KUKA KRL program: Robotica_Trabalho_v4.src, Robotica_Trabalho_v4.dat

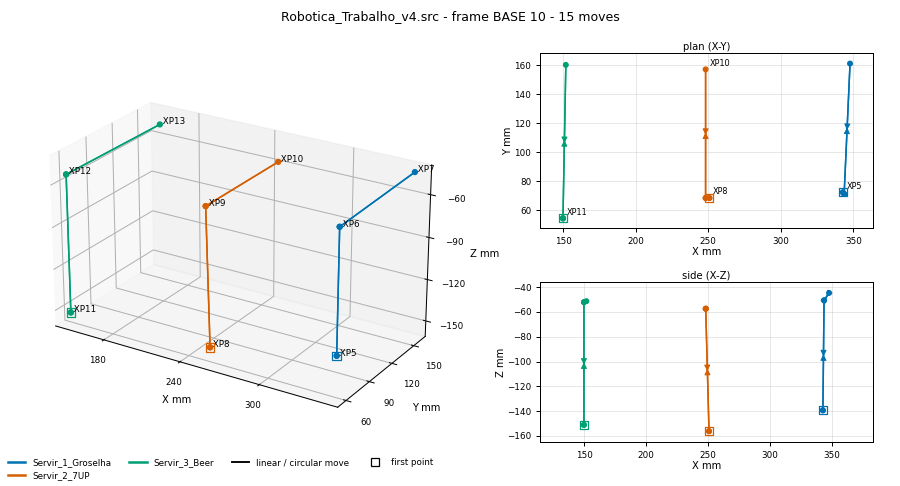
[picture p0: tool path of Robotica_Trabalho_v4.src in frame BASE 10, 15 of 36 moves have a stored position in this frame; points joined in program order, loops and branches not executed]
--- Robotica_Trabalho_v4.src ---
&ACCESS RVP
&REL 213
&PARAM DISKPATH = KRC:\R1\Program\meec2021\G3
DEF Robotica_Trabalho_v3( )
;FOLD INI
  ;FOLD BASISTECH INI
    GLOBAL INTERRUPT DECL 3 WHEN $STOPMESS==TRUE DO IR_STOPM ( )
    INTERRUPT ON 3
    BAS (#INITMOV,0 )
  ;ENDFOLD (BASISTECH INI)
  ;FOLD USER INI
    ;Make your modifications here

  ;ENDFOLD (USER INI)
;ENDFOLD (INI)
$ADVANCE=0


flag_Cycle_Copos = FALSE ;Quando usar 3 copos, passa a TRUE e para o robô

GLOBAL INTERRUPT DECL 1 WHEN flag_Cycle_Copos==TRUE DO StopProg()

;ponto para o sistema de visao
G3_sistema_visao = {X 0,Y 0,Z 23.56,A 93.23,B 1.40,C 0}

XG3_HOME = {X 593.30,Y -262.56,Z 438.69,A 6.37,B 2.12,C 1.97,S 6,T 18,E1 0.0,E2 0.0,E3 0.0,E4 0.0,E5 0.0,E6 0.0}
;FOLD PTP G3_HOME CONT Vel=100 % PDAT7 Tool[5]:G3_COPO Base[0];%{PE}%R 8.2.24,%MKUKATPBASIS,%CMOVE,%VPTP,%P 1:PTP, 2:G3_HOME, 3:C_DIS, 5:100, 7:PDAT7
$BWDSTART=FALSE
PDAT_ACT=PPDAT7
FDAT_ACT=FG3_HOME
BAS(#PTP_PARAMS,100)
PTP XG3_HOME C_DIS
;ENDFOLD

;**************************************
;       Set Variables
;**************************************
NUM_COPO = 3
NUM_PORTIONS_1= 0
NUM_PORTIONS_2 = 0
NUM_PORTIONS_3 = 0
Flag_Tirar_Bebida = FALSE
Flag_Arrumar_Copo = FALSE

INTERRUPT ON
INTERRUPT ENABLE


flag_Cycle_Copos = TRUE
aux_func()

LOOP


IF Flag_Tirar_Bebida == TRUE THEN

PegarCopo(NUM_COPO)
Servir_1_Groselha(NUM_PORTIONS_1)
Servir_2_7UP(NUM_PORTIONS_2)
Servir_3_Beer(NUM_PORTIONS_3)

;FOLD PTP G3_HOME CONT Vel=100 % PDAT19 Tool[5]:G3_COPO Base[0];%{PE}%R 8.2.24,%MKUKATPBASIS,%CMOVE,%VPTP,%P 1:PTP, 2:G3_HOME, 3:C_DIS, 5:100, 7:PDAT19
$BWDSTART=FALSE
PDAT_ACT=PPDAT19
FDAT_ACT=FG3_HOME
BAS(#PTP_PARAMS,100)
PTP XG3_HOME C_DIS
;ENDFOLD
Entrega_Bebida(NUM_COPO)

NUM_COPO = NUM_COPO - 1
Flag_Tirar_Bebida = FALSE

ENDIF

IF Flag_Arrumar_Copo == TRUE THEN

ArrumarCopo()  ;Pega no copo usado para lavar
Flag_Arrumar_Copo = FALSE

ENDIF

ENDLOOP

;FOLD PTP G3_HOME  Vel=100 % PDAT8 Tool[5] Base[0];%{PE}%R 8.2.17,%MKUKATPBASIS,%CMOVE,%VPTP,%P 1:PTP, 2:G3_HOME, 3:, 5:100, 7:PDAT8
$BWDSTART=FALSE
PDAT_ACT=PPDAT8
FDAT_ACT=FG3_HOME
BAS(#PTP_PARAMS,100)
PTP XG3_HOME
;ENDFOLD


END
;***********************************************
;  Função responsável por pegar num copo Novo
;***********************************************
DEF PegarCopo(NUM_COPO:in)
INT NUM_COPO
;INT aux=0


IF (NUM_COPO > 0) AND (NUM_COPO < 4) THEN  ;Se for utilizados 3 copos não vai buscar o 4º

SWITCH NUM_COPO
CASE 3
aux =1 ;nao faz shift
CASE 2
aux = 2  ;shift do copo 2
CASE 1
aux = 3  ;shift do copo 3
DEFAULT
ENDSWITCH

;FOLD OUT 1 'close' State=FALSE CONT;%{PE}%R 8.2.24,%MKUKATPBASIS,%COUT,%VOUTX,%P 2:1, 3:close, 5:FALSE, 6:CONTINUE
CONTINUE
$OUT[1]=FALSE
;ENDFOLD
;FOLD OUT 4 'open' State=FALSE CONT;%{PE}%R 8.2.24,%MKUKATPBASIS,%COUT,%VOUTX,%P 2:4, 3:open, 5:FALSE, 6:CONTINUE
CONTINUE
$OUT[4]=FALSE
;ENDFOLD

;Posiciona o gripper paralelo com o copo mas num ponto mais alto
;FOLD PTP P1 CONT Vel=100 % PDAT1 Tool[5]:G3_COPO Base[9]:meec21_G3_copos;%{PE}%R 8.2.24,%MKUKATPBASIS,%CMOVE,%VPTP,%P 1:PTP, 2:P1, 3:C_DIS, 5:100, 7:PDAT1
$BWDSTART=FALSE
PDAT_ACT=PPDAT1
FDAT_ACT=FP1
BAS(#PTP_PARAMS,100)
PTP XP1 C_DIS
;ENDFOLD

;Abre o Gripper
;FOLD OUT 4 'open' State=TRUE CONT;%{PE}%R 8.2.24,%MKUKATPBASIS,%COUT,%VOUTX,%P 2:4, 3:open, 5:TRUE, 6:CONTINUE
CONTINUE
$OUT[4]=TRUE
;ENDFOLD
;FOLD WAIT Time=0.1 sec;%{PE}%R 8.2.24,%MKUKATPBASIS,%CWAIT,%VWAIT,%P 3:0.1
WAIT SEC 0.1
;ENDFOLD
;FOLD OUT 4 'open' State=FALSE CONT;%{PE}%R 8.2.24,%MKUKATPBASIS,%COUT,%VOUTX,%P 2:4, 3:open, 5:FALSE, 6:CONTINUE
CONTINUE
$OUT[4]=FALSE
;ENDFOLD

;Posiciona o Gripper paralelo com o copo
;FOLD LIN P2 CONT Vel=2 m/s CPDAT1 Tool[5]:G3_COPO Base[9]:meec21_G3_copos;%{PE}%R 8.2.24,%MKUKATPBASIS,%CMOVE,%VLIN,%P 1:LIN, 2:P2, 3:C_DIS C_DIS, 5:2, 7:CPDAT1
$BWDSTART=FALSE
LDAT_ACT=LCPDAT1
FDAT_ACT=FP2
BAS(#CP_PARAMS,2)
LIN XP2 C_DIS C_DIS
;ENDFOLD

;Posiciona o copo dentro da pinça

XP3={X 197.8517,Y 191.609207,Z 11.5482101,A 92.7861786,B 4.34509897,C 2.74875402}:Shift_Copo[aux]
;FOLD LIN P3 CONT Vel=2 m/s CPDAT2 Tool[5]:G3_COPO Base[9]:meec21_G3_copos;%{PE}%R 8.2.24,%MKUKATPBASIS,%CMOVE,%VLIN,%P 1:LIN, 2:P3, 3:C_DIS C_DIS, 5:2, 7:CPDAT2
$BWDSTART=FALSE
LDAT_ACT=LCPDAT2
FDAT_ACT=FP3
BAS(#CP_PARAMS,2)
LIN XP3 C_DIS C_DIS
;ENDFOLD


;Fecha o Gripper
;FOLD OUT 1 'close' State=TRUE CONT;%{PE}%R 8.2.24,%MKUKATPBASIS,%COUT,%VOUTX,%P 2:1, 3:close, 5:TRUE, 6:CONTINUE
CONTINUE
$OUT[1]=TRUE
;ENDFOLD
;FOLD WAIT Time=0.1 sec;%{PE}%R 8.2.24,%MKUKATPBASIS,%CWAIT,%VWAIT,%P 3:0.1
WAIT SEC 0.1
;ENDFOLD
;FOLD OUT 1 'close' State=FALSE CONT;%{PE}%R 8.2.24,%MKUKATPBASIS,%COUT,%VOUTX,%P 2:1, 3:close, 5:FALSE, 6:CONTINUE
CONTINUE
$OUT[1]=FALSE
;ENDFOLD


;Levanta o copo num movimento vertical
XP4={X 197.849304,Y 191.610901,Z 204.555206,A 92.7863464,B 4.34535694,C 2.74913096}:Shift_Copo[aux]
;FOLD LIN P4 CONT Vel=2 m/s CPDAT3 Tool[5]:G3_COPO Base[9]:meec21_G3_copos;%{PE}%R 8.2.24,%MKUKATPBASIS,%CMOVE,%VLIN,%P 1:LIN, 2:P4, 3:C_DIS C_DIS, 5:2, 7:CPDAT3
$BWDSTART=FALSE
LDAT_ACT=LCPDAT3
FDAT_ACT=FP4
BAS(#CP_PARAMS,2)
LIN XP4 C_DIS C_DIS
;ENDFOLD



ELSE
flag_Cycle_Copos = TRUE  ;Irá lançar um interrupção e parar o programa até a flag voltar a FALSE

ENDIF

END
;****************************************************
;  Função Responsável por despejar uma porcao de Groselha
;*******************************************
DEF Servir_1_Groselha(NUM_Por:IN)
INT NUM_Por

IF NUM_Por > 0 THEN

;Posiciona o gripper alinhado com a zona da bebida mas longe da garrafa
;FOLD PTP P5 CONT Vel=100 % PDAT2 Tool[5]:G3_COPO Base[10]:meec_G3_bebidas;%{PE}%R 8.2.24,%MKUKATPBASIS,%CMOVE,%VPTP,%P 1:PTP, 2:P5, 3:C_DIS, 5:100, 7:PDAT2
$BWDSTART=FALSE
PDAT_ACT=PPDAT2
FDAT_ACT=FP5
BAS(#PTP_PARAMS,100)
PTP XP5 C_DIS
;ENDFOLD

;Posiciona-se debaixo da garrafa de Groselha
;FOLD LIN P6 CONT Vel=1 m/s CPDAT6 Tool[5]:G3_COPO Base[10]:meec_G3_bebidas;%{PE}%R 8.2.24,%MKUKATPBASIS,%CMOVE,%VLIN,%P 1:LIN, 2:P6, 3:C_DIS C_DIS, 5:1, 7:CPDAT6
$BWDSTART=FALSE
LDAT_ACT=LCPDAT6
FDAT_ACT=FP6
BAS(#CP_PARAMS,1)
LIN XP6 C_DIS C_DIS
;ENDFOLD

FOR i = NUM_Por TO 1 STEP -1

;Faz força contra o doseador para começar a despejar
;FOLD LIN P7 CONT Vel=0.4 m/s CPDAT5 Tool[5]:G3_COPO Base[10]:meec_G3_bebidas;%{PE}%R 8.2.24,%MKUKATPBASIS,%CMOVE,%VLIN,%P 1:LIN, 2:P7, 3:C_DIS C_DIS, 5:0.4, 7:CPDAT5
$BWDSTART=FALSE
LDAT_ACT=LCPDAT5
FDAT_ACT=FP7
BAS(#CP_PARAMS,0.4)
LIN XP7 C_DIS C_DIS
;ENDFOLD
;Espera 1,5 segundos para o doseador despejar no copo
;FOLD WAIT Time=3 sec;%{PE}%R 8.2.24,%MKUKATPBASIS,%CWAIT,%VWAIT,%P 3:3
WAIT SEC 3
;ENDFOLD
;FOLD LIN P6 CONT Vel=1 m/s CPDAT0 Tool[5]:G3_COPO Base[10]:meec_G3_bebidas;%{PE}%R 8.2.24,%MKUKATPBASIS,%CMOVE,%VLIN,%P 1:LIN, 2:P6, 3:C_DIS C_DIS, 5:1, 7:CPDAT0
$BWDSTART=FALSE
LDAT_ACT=LCPDAT0
FDAT_ACT=FP6
BAS(#CP_PARAMS,1)
LIN XP6 C_DIS C_DIS
;ENDFOLD

IF NUM_Por > 1 THEN
;Espera uns segundos para voltar a encher o doseador se a bebida tiver mais do que uma dose da mesma bebida
;FOLD WAIT Time= 3 sec;%{PE}%R 8.3.22,%MKUKATPBASIS,%CWAIT,%VWAIT,%P 2:3
WAIT SEC 3
;ENDFOLD
ENDIF

ENDFOR

;FOLD LIN P5 CONT Vel=1 m/s CPDAT7 Tool[5]:G3_COPO Base[10]:meec_G3_bebidas;%{PE}%R 8.2.24,%MKUKATPBASIS,%CMOVE,%VLIN,%P 1:LIN, 2:P5, 3:C_DIS C_DIS, 5:1, 7:CPDAT7
$BWDSTART=FALSE
LDAT_ACT=LCPDAT7
FDAT_ACT=FP5
BAS(#CP_PARAMS,1)
LIN XP5 C_DIS C_DIS
;ENDFOLD

ENDIF

END
;**********************************************
;  Função Responsável por despejar uma porcao de 7Up
;**********************************************
DEF Servir_2_7UP(NUM_Por :IN)
INT NUM_Por

IF NUM_Por > 0 THEN

;FOLD PTP P8 CONT Vel=100 % PDAT5 Tool[5]:G3_COPO Base[10]:meec_G3_bebidas;%{PE}%R 8.2.24,%MKUKATPBASIS,%CMOVE,%VPTP,%P 1:PTP, 2:P8, 3:C_DIS, 5:100, 7:PDAT5
$BWDSTART=FALSE
PDAT_ACT=PPDAT5
FDAT_ACT=FP8
BAS(#PTP_PARAMS,100)
PTP XP8 C_DIS
;ENDFOLD

;FOLD LIN P9 CONT Vel=1 m/s CPDAT8 Tool[5]:G3_COPO Base[10]:meec_G3_bebidas;%{PE}%R 8.2.24,%MKUKATPBASIS,%CMOVE,%VLIN,%P 1:LIN, 2:P9, 3:C_DIS C_DIS, 5:1, 7:CPDAT8
$BWDSTART=FALSE
LDAT_ACT=LCPDAT8
FDAT_ACT=FP9
BAS(#CP_PARAMS,1)
LIN XP9 C_DIS C_DIS
;ENDFOLD

FOR i=NUM_Por TO 1 STEP -1

;FOLD LIN P10 CONT Vel=0.4 m/s CPDAT9 Tool[5]:G3_COPO Base[10]:meec_G3_bebidas;%{PE}%R 8.2.24,%MKUKATPBASIS,%CMOVE,%VLIN,%P 1:LIN, 2:P10, 3:C_DIS C_DIS, 5:0.4, 7:CPDAT9
$BWDSTART=FALSE
LDAT_ACT=LCPDAT9
FDAT_ACT=FP10
BAS(#CP_PARAMS,0.4)
LIN XP10 C_DIS C_DIS
;ENDFOLD

;FOLD WAIT 1.5 3 sec;%{PE}%R 8.2.24,%MKUKATPBASIS,%CWAIT,%VWAIT,%P 3:3
WAIT SEC 3
;ENDFOLD

;FOLD LIN P9 CONT Vel=1 m/s CPDAT10 Tool[5]:G3_COPO Base[10]:meec_G3_bebidas;%{PE}%R 8.2.24,%MKUKATPBASIS,%CMOVE,%VLIN,%P 1:LIN, 2:P9, 3:C_DIS C_DIS, 5:1, 7:CPDAT10
$BWDSTART=FALSE
LDAT_ACT=LCPDAT10
FDAT_ACT=FP9
BAS(#CP_PARAMS,1)
LIN XP9 C_DIS C_DIS
;ENDFOLD

IF NUM_Por > 1 THEN
;FOLD WAIT Time= 3 sec;%{PE}%R 8.3.22,%MKUKATPBASIS,%CWAIT,%VWAIT,%P 2:3
WAIT SEC 3
;ENDFOLD
ENDIF

ENDFOR

;FOLD LIN P8 CONT Vel=1 m/s CPDAT11 Tool[5]:G3_COPO Base[10]:meec_G3_bebidas;%{PE}%R 8.2.24,%MKUKATPBASIS,%CMOVE,%VLIN,%P 1:LIN, 2:P8, 3:C_DIS C_DIS, 5:1, 7:CPDAT11
$BWDSTART=FALSE
LDAT_ACT=LCPDAT11
FDAT_ACT=FP8
BAS(#CP_PARAMS,1)
LIN XP8 C_DIS C_DIS
;ENDFOLD

ENDIF

END
;************************************************
;  Função Responsável por despejar uma porcao de Cerveja
;************************************************
DEF Servir_3_Beer(NUM_Por :IN)
INT NUM_Por

IF NUM_Por > 0 THEN

;FOLD PTP P11 CONT Vel=100 % PDAT6 Tool[5]:G3_COPO Base[10]:meec_G3_bebidas;%{PE}%R 8.2.24,%MKUKATPBASIS,%CMOVE,%VPTP,%P 1:PTP, 2:P11, 3:C_DIS, 5:100, 7:PDAT6
$BWDSTART=FALSE
PDAT_ACT=PPDAT6
FDAT_ACT=FP11
BAS(#PTP_PARAMS,100)
PTP XP11 C_DIS
;ENDFOLD

;FOLD LIN P12 CONT Vel=1 m/s CPDAT12 Tool[5]:G3_COPO Base[10]:meec_G3_bebidas;%{PE}%R 8.2.24,%MKUKATPBASIS,%CMOVE,%VLIN,%P 1:LIN, 2:P12, 3:C_DIS C_DIS, 5:1, 7:CPDAT12
$BWDSTART=FALSE
LDAT_ACT=LCPDAT12
FDAT_ACT=FP12
BAS(#CP_PARAMS,1)
LIN XP12 C_DIS C_DIS
;ENDFOLD

FOR i=NUM_Por TO 1 STEP -1
;FOLD LIN P13 CONT Vel=0.4 m/s CPDAT13 Tool[5]:G3_COPO Base[10]:meec_G3_bebidas;%{PE}%R 8.2.24,%MKUKATPBASIS,%CMOVE,%VLIN,%P 1:LIN, 2:P13, 3:C_DIS C_DIS, 5:0.4, 7:CPDAT13
$BWDSTART=FALSE
LDAT_ACT=LCPDAT13
FDAT_ACT=FP13
BAS(#CP_PARAMS,0.4)
LIN XP13 C_DIS C_DIS
;ENDFOLD
;FOLD WAIT 1.5 3 sec;%{PE}%R 8.2.24,%MKUKATPBASIS,%CWAIT,%VWAIT,%P 3:3
WAIT SEC 3
;ENDFOLD

;FOLD LIN P12 CONT Vel=1 m/s CPDAT14 Tool[5]:G3_COPO Base[10]:meec_G3_bebidas;%{PE}%R 8.2.24,%MKUKATPBASIS,%CMOVE,%VLIN,%P 1:LIN, 2:P12, 3:C_DIS C_DIS, 5:1, 7:CPDAT14
$BWDSTART=FALSE
LDAT_ACT=LCPDAT14
FDAT_ACT=FP12
BAS(#CP_PARAMS,1)
LIN XP12 C_DIS C_DIS
;ENDFOLD

IF NUM_Por > 1 THEN
;FOLD WAIT Time= 3 sec;%{PE}%R 8.3.22,%MKUKATPBASIS,%CWAIT,%VWAIT,%P 2:3
WAIT SEC 3
;ENDFOLD
ENDIF

ENDFOR

;FOLD LIN P11 CONT Vel=1 m/s CPDAT15 Tool[5]:G3_COPO Base[10]:meec_G3_bebidas;%{PE}%R 8.3.22,%MKUKATPBASIS,%CMOVE,%VLIN,%P 1:LIN, 2:P11, 3:C_DIS C_DIS, 5:1, 7:CPDAT15
$BWDSTART=FALSE
LDAT_ACT=LCPDAT15
FDAT_ACT=FP11
BAS(#CP_PARAMS,1)
LIN XP11 C_DIS C_DIS
;ENDFOLD

ENDIF

END
;************************************
; Função para entregar copo com bebida
;************************************
DEF Entrega_Bebida(NUM_COPO:in)
INT NUM_COPO

IF (NUM_COPO > 0) AND (NUM_COPO < 4) THEN  ;Certifica-se que são apenas 3 copos

SWITCH NUM_COPO
CASE 3
aux =1 ;nao faz shift
CASE 2
aux = 2  ;shift do copo 2
CASE 1
aux = 3  ;shift do copo 3
DEFAULT
ENDSWITCH

;Posiciona-se em cima do ponto de pousar o copo
XP14={X 367.326996,Y 369.67511,Z 89.1293869,A 96.3636475,B 4.65242004,C 2.64675307}:Shift_Entregar_Copo[aux]
;FOLD PTP P14 CONT Vel=100 % PDAT2 Tool[5]:G3_COPO Base[9]:meec21_G3_copos;%{PE}%R 8.2.24,%MKUKATPBASIS,%CMOVE,%VPTP,%P 1:PTP, 2:P14, 3:C_DIS, 5:100, 7:PDAT2
$BWDSTART=FALSE
PDAT_ACT=PPDAT2
FDAT_ACT=FP14
BAS(#PTP_PARAMS,100)
PTP XP14 C_DIS
;ENDFOLD

;Posiciona o copo na zona onde o irá largar
XP15={X 363.682404,Y 361.287598,Z -8.55531788,A 96.3680573,B 4.63769197,C 2.64578199}:Shift_Entregar_Copo[aux]
;FOLD LIN P15 CONT Vel=1 m/s CPDAT3 Tool[5]:G3_COPO Base[9]:meec21_G3_copos;%{PE}%R 8.2.24,%MKUKATPBASIS,%CMOVE,%VLIN,%P 1:LIN, 2:P15, 3:C_DIS C_DIS, 5:1, 7:CPDAT3
$BWDSTART=FALSE
LDAT_ACT=LCPDAT3
FDAT_ACT=FP15
BAS(#CP_PARAMS,1)
LIN XP15 C_DIS C_DIS
;ENDFOLD

;Abre o Gripper
;FOLD OUT 4 'open' State=TRUE CONT;%{PE}%R 8.2.24,%MKUKATPBASIS,%COUT,%VOUTX,%P 2:4, 3:open, 5:TRUE, 6:CONTINUE
CONTINUE
$OUT[4]=TRUE
;ENDFOLD
;FOLD WAIT Time=0.1 sec;%{PE}%R 8.2.24,%MKUKATPBASIS,%CWAIT,%VWAIT,%P 3:0.1
WAIT SEC 0.1
;ENDFOLD
;FOLD OUT 4 'open' State=FALSE CONT;%{PE}%R 8.2.24,%MKUKATPBASIS,%COUT,%VOUTX,%P 2:4, 3:open, 5:FALSE, 6:CONTINUE
CONTINUE
$OUT[4]=FALSE
;ENDFOLD

;Move para o lado de modo ao copo sair do Gripper
XP16={X 365.064514,Y 281.376587,Z 1.60763502,A 96.368042,B 4.63726902,C 2.6456461}:Shift_Entregar_Copo[aux]
;FOLD LIN P16 CONT Vel=1 m/s CPDAT4 Tool[5]:G3_COPO Base[9]:meec21_G3_copos;%{PE}%R 8.2.24,%MKUKATPBASIS,%CMOVE,%VLIN,%P 1:LIN, 2:P16, 3:C_DIS C_DIS, 5:1, 7:CPDAT4
$BWDSTART=FALSE
LDAT_ACT=LCPDAT4
FDAT_ACT=FP16
BAS(#CP_PARAMS,1)
LIN XP16 C_DIS C_DIS
;ENDFOLD

;Levanta o Gripper
XP17={X 368.319214,Y 288.928009,Z 89.7433701,A 96.368721,B 4.63736916,C 2.64742398}:Shift_Entregar_Copo[aux]
;FOLD LIN P17 CONT Vel=1 m/s CPDAT5 Tool[5]:G3_COPO Base[9]:meec21_G3_copos;%{PE}%R 8.2.24,%MKUKATPBASIS,%CMOVE,%VLIN,%P 1:LIN, 2:P17, 3:C_DIS C_DIS, 5:1, 7:CPDAT5
$BWDSTART=FALSE
LDAT_ACT=LCPDAT5
FDAT_ACT=FP17
BAS(#CP_PARAMS,1)
LIN XP17 C_DIS C_DIS
;ENDFOLD

;FOLD PTP G3_HOME CONT Vel=100 % PDAT22 Tool[5]:G3_COPO Base[0];%{PE}%R 8.2.24,%MKUKATPBASIS,%CMOVE,%VPTP,%P 1:PTP, 2:G3_HOME, 3:C_DIS, 5:100, 7:PDAT22
$BWDSTART=FALSE
PDAT_ACT=PPDAT22
FDAT_ACT=FG3_HOME
BAS(#PTP_PARAMS,100)
PTP XG3_HOME C_DIS
;ENDFOLD

ENDIF

END
;*******************************
;  Arruma copo usado
;*******************************
DEF ArrumarCopo()

;Abre o Gripper
;FOLD OUT 4 'open' State=TRUE CONT;%{PE}%R 8.2.24,%MKUKATPBASIS,%COUT,%VOUTX,%P 2:4, 3:open, 5:TRUE, 6:CONTINUE
CONTINUE
$OUT[4]=TRUE
;ENDFOLD
;FOLD WAIT Time=0.1 sec;%{PE}%R 8.2.24,%MKUKATPBASIS,%CWAIT,%VWAIT,%P 3:0.1
WAIT SEC 0.1
;ENDFOLD
;FOLD OUT 4 'open' State=FALSE CONT;%{PE}%R 8.2.24,%MKUKATPBASIS,%COUT,%VOUTX,%P 2:4, 3:open, 5:FALSE, 6:CONTINUE
CONTINUE
$OUT[4]=FALSE
;ENDFOLD

;Posiciona a tool num ponto atras e em cima
;FOLD PTP G3_sistema_visao CONT Vel=100 % PDAT13 Tool[5]:G3_COPO Base[11]:G3_Visao;%{PE}%R 8.2.24,%MKUKATPBASIS,%CMOVE,%VPTP,%P 1:PTP, 2:G3_sistema_visao, 3:C_DIS, 5:100, 7:PDAT13
$BWDSTART=FALSE
PDAT_ACT=PPDAT13
FDAT_ACT=FG3_sistema_visao
BAS(#PTP_PARAMS,100)
PTP XG3_sistema_visao C_DIS
;ENDFOLD
XP18 = G3_sistema_visao:Shift_Copo_Sujo[1]
;FOLD PTP P18 CONT Vel=100 % PDAT3 Tool[5]:G3_COPO Base[11]:G3_Visao;%{PE}%R 8.2.24,%MKUKATPBASIS,%CMOVE,%VPTP,%P 1:PTP, 2:P18, 3:C_DIS, 5:100, 7:PDAT3
$BWDSTART=FALSE
PDAT_ACT=PPDAT3
FDAT_ACT=FP18
BAS(#PTP_PARAMS,100)
PTP XP18 C_DIS
;ENDFOLD

;Posiciona a tool atras do copo
XP19 = G3_sistema_visao:Shift_Copo_Sujo[2]
;FOLD LIN P19 CONT Vel=1 m/s CPDAT6 Tool[5]:G3_COPO Base[11]:G3_Visao;%{PE}%R 8.2.24,%MKUKATPBASIS,%CMOVE,%VLIN,%P 1:LIN, 2:P19, 3:C_DIS C_DIS, 5:1, 7:CPDAT6
$BWDSTART=FALSE
LDAT_ACT=LCPDAT6
FDAT_ACT=FP19
BAS(#CP_PARAMS,1)
LIN XP19 C_DIS C_DIS
;ENDFOLD

;Posição do copo recebida pelo PC
XP20 = G3_sistema_visao:Shift_Copo_Sujo[3]
;FOLD LIN P20 Vel=1 m/s CPDAT7 Tool[5]:G3_COPO Base[11]:G3_Visao;%{PE}%R 8.2.24,%MKUKATPBASIS,%CMOVE,%VLIN,%P 1:LIN, 2:P20, 3:, 5:1, 7:CPDAT7
$BWDSTART=FALSE
LDAT_ACT=LCPDAT7
FDAT_ACT=FP20
BAS(#CP_PARAMS,1)
LIN XP20
;ENDFOLD

;Fecha o Gripper
;FOLD OUT 1 'close' State=TRUE CONT;%{PE}%R 8.2.24,%MKUKATPBASIS,%COUT,%VOUTX,%P 2:1, 3:close, 5:TRUE, 6:CONTINUE
CONTINUE
$OUT[1]=TRUE
;ENDFOLD
;FOLD WAIT Time=0.1 sec;%{PE}%R 8.2.24,%MKUKATPBASIS,%CWAIT,%VWAIT,%P 3:0.1
WAIT SEC 0.1
;ENDFOLD
;FOLD OUT 1 'close' State=FALSE CONT;%{PE}%R 8.2.24,%MKUKATPBASIS,%COUT,%VOUTX,%P 2:1, 3:close, 5:FALSE, 6:CONTINUE
CONTINUE
$OUT[1]=FALSE
;ENDFOLD

;Posição a cima do copo
XP21 = G3_sistema_visao:Shift_Copo_Sujo[4]
;FOLD LIN P21 CONT Vel=1 m/s CPDAT8 Tool[5]:G3_COPO Base[11]:G3_Visao;%{PE}%R 8.2.24,%MKUKATPBASIS,%CMOVE,%VLIN,%P 1:LIN, 2:P21, 3:C_DIS C_DIS, 5:1, 7:CPDAT8
$BWDSTART=FALSE
LDAT_ACT=LCPDAT8
FDAT_ACT=FP21
BAS(#CP_PARAMS,1)
LIN XP21 C_DIS C_DIS
;ENDFOLD

;Posciona o copo em cima do lixo
;FOLD PTP P22 CONT Vel=100 % PDAT4 Tool[5]:G3_COPO Base[11]:G3_Visao;%{PE}%R 8.2.24,%MKUKATPBASIS,%CMOVE,%VPTP,%P 1:PTP, 2:P22, 3:C_DIS, 5:100, 7:PDAT4
$BWDSTART=FALSE
PDAT_ACT=PPDAT4
FDAT_ACT=FP22
BAS(#PTP_PARAMS,100)
PTP XP22 C_DIS
;ENDFOLD

;Abre o Gripper
;FOLD OUT 4 'open' State=TRUE CONT;%{PE}%R 8.2.24,%MKUKATPBASIS,%COUT,%VOUTX,%P 2:4, 3:open, 5:TRUE, 6:CONTINUE
CONTINUE
$OUT[4]=TRUE
;ENDFOLD
;FOLD WAIT Time=0.1 sec;%{PE}%R 8.2.24,%MKUKATPBASIS,%CWAIT,%VWAIT,%P 3:0.1
WAIT SEC 0.1
;ENDFOLD
;FOLD OUT 4 'open' State=FALSE CONT;%{PE}%R 8.2.24,%MKUKATPBASIS,%COUT,%VOUTX,%P 2:4, 3:open, 5:FALSE, 6:CONTINUE
CONTINUE
$OUT[4]=FALSE
;ENDFOLD

;FOLD PTP G3_HOME CONT Vel=100 % PDAT14 Tool[5]:G3_COPO Base[0];%{PE}%R 8.2.24,%MKUKATPBASIS,%CMOVE,%VPTP,%P 1:PTP, 2:G3_HOME, 3:C_DIS, 5:100, 7:PDAT14
$BWDSTART=FALSE
PDAT_ACT=PPDAT14
FDAT_ACT=FG3_HOME
BAS(#PTP_PARAMS,100)
PTP XG3_HOME C_DIS
;ENDFOLD

END

;*************************************
; Função para Parar o robô quando usar mais do que 3 copos
;*************************************
DEF StopProg()
INTERRUPT OFF
;REPEAT  ;Repete este ciclo ate flag = TRUE

;FOLD PTP G3_HOME CONT Vel=100 % PDAT20 Tool[5]:G3_COPO Base[0];%{PE}%R 8.2.24,%MKUKATPBASIS,%CMOVE,%VPTP,%P 1:PTP, 2:G3_HOME, 3:C_DIS, 5:100, 7:PDAT20
$BWDSTART=FALSE
PDAT_ACT=PPDAT20
FDAT_ACT=FG3_HOME
BAS(#PTP_PARAMS,100)
PTP XG3_HOME C_DIS
;ENDFOLD

;FOLD PTP HOME CONT Vel=100 % PDAT21;%{PE}%R 8.2.24,%MKUKATPBASIS,%CMOVE,%VPTP,%P 1:PTP, 2:HOME, 3:C_DIS, 5:100, 7:PDAT21
$BWDSTART=FALSE
PDAT_ACT=PPDAT21
FDAT_ACT=FHOME
BAS(#PTP_PARAMS,100)
$H_POS=XHOME
PTP XHOME C_DIS
;ENDFOLD
;UNTIL flag_Cycle_Copos == FALSE

;NUM_COPO = 3 ;numero de copos restantes, declarado como external no ficheiro .dat5
RESUME
END
;*******************************
;  DECLARA OS SHISFTS DE POSIÇÃO
;*******************************
DEF aux_func()

Shift_Copo[1] = {X 0,Y 0,Z 0,A 0,B 0,C 0} ;1 copo, nao faz shift
Shift_Copo[2] = {X 89.95,Y 0,Z 0,A 0,B 0,C 0} ;shift de pegar 2 copo
Shift_Copo[3] = {X 174.341, Y -2.617,Z 0,A 0,B 0, C 0} ;shift de pegar 3 copo

Shift_Entregar_Copo[1] = {X 0,Y 0,Z 0,A 0,B 0,C 0}
Shift_Entregar_Copo[2] = {X -78,Y 10,Z 0,A 0,B 0,C 0}
Shift_Entregar_Copo[3] = {X -164.341,Y 15,Z 20,A 0,B 0,C 0}


;Shits referentes a pegar no copo e levar para valar
Shift_Copo_Sujo[1] = {X -60,Y -36,Z 200,A 0,B 0,C 0};
Shift_Copo_Sujo[2] = {X -60,Y -36,Z 20,A 0,B 0,C 0};
Shift_Copo_Sujo[3] = {X 20,Y -36,Z 20,A 0,B 0,C 0};
Shift_Copo_Sujo[4] = {X 0,Y -36,Z 200,A 0,B 0,C 0};

;Inserir os valores corretos das coordenadas do shift

END

--- Robotica_Trabalho_v4.dat ---
&ACCESS RVP
&REL 213
&PARAM DISKPATH = KRC:\R1\Program\meec2021\G3
DEFDAT  Robotica_Trabalho_v3 PUBLIC
;FOLD EXTERNAL DECLARATIONS;%{PE}%MKUKATPBASIS,%CEXT,%VCOMMON,%P
;FOLD BASISTECH EXT;%{PE}%MKUKATPBASIS,%CEXT,%VEXT,%P
EXT  BAS (BAS_COMMAND  :IN,REAL  :IN )
DECL INT SUCCESS
;ENDFOLD (BASISTECH EXT)
;FOLD USER EXT;%{E}%MKUKATPUSER,%CEXT,%VEXT,%P
;Make here your modifications
DECL INT NUM_COPO
DECL E6POS Shift_Copo[3]
DECL E6POS Shift_Entregar_Copo[3]
DECL E6POS Shift_Copo_Sujo[4]
DECL BOOL flag_Cycle_Copos
DECL INT aux

;ENDFOLD (USER EXT)
;ENDFOLD (EXTERNAL DECLERATIONS)
DECL BASIS_SUGG_T LAST_BASIS={POINT1[] "G3_HOME                 ",POINT2[] "G3_HOME                 ",CP_PARAMS[] "CPDAT8                  ",PTP_PARAMS[] "PDAT22                  ",CONT[] "C_DIS                   ",CP_VEL[] "0.4                     ",PTP_VEL[] "100                     ",SYNC_PARAMS[] "SYNCDAT                 ",SPL_NAME[] "S0                      "}
DECL E6POS XP11={X 149.957596,Y 54.5289688,Z -151.048203,A -34.5448189,B -88.7538681,C -53.1429596,S 6,T 18,E1 0.0,E2 0.0,E3 0.0,E4 0.0,E5 0.0,E6 0.0}
DECL FDAT FP11={TOOL_NO 5,BASE_NO 10,IPO_FRAME #BASE,POINT2[] " ",TQ_STATE FALSE}
DECL PDAT PPDAT6={VEL 100.0,ACC 100.0,APO_DIST 100.0,APO_MODE #CDIS,GEAR_JERK 50.0}
DECL E6POS XP12={X 149.958694,Y 54.5240784,Z -52.0914001,A -34.5103188,B -88.7544327,C -53.1793709,S 6,T 18,E1 0.0,E2 0.0,E3 0.0,E4 0.0,E5 0.0,E6 0.0}
DECL FDAT FP12={TOOL_NO 5,BASE_NO 10,IPO_FRAME #BASE,POINT2[] " ",TQ_STATE FALSE}
DECL LDAT LCPDAT12={VEL 2.0,ACC 100.0,APO_DIST 100.0,APO_FAC 50.0,AXIS_VEL 100.0,AXIS_ACC 100.0,ORI_TYP #VAR,CIRC_TYP #BASE,JERK_FAC 50.0,GEAR_JERK 50.0,EXAX_IGN 0}
DECL LDAT LCPDAT15={VEL 2.0,ACC 100.0,APO_DIST 100.0,APO_FAC 50.0,AXIS_VEL 100.0,AXIS_ACC 100.0,ORI_TYP #VAR,CIRC_TYP #BASE,JERK_FAC 50.0,GEAR_JERK 50.0,EXAX_IGN 0}
DECL E6POS XP1={X 200.690094,Y 97.6676102,Z 212.382904,A 92.7856369,B 4.34229183,C 2.74763393,S 6,T 18,E1 0.0,E2 0.0,E3 0.0,E4 0.0,E5 0.0,E6 0.0}
DECL FDAT FP1={TOOL_NO 5,BASE_NO 9,IPO_FRAME #BASE,POINT2[] " ",TQ_STATE FALSE}
DECL PDAT PPDAT1={VEL 100.0,ACC 100.0,APO_DIST 100.0,APO_MODE #CDIS}
DECL E6POS XP2={X 198.5569,Y 108.492401,Z 11.5661201,A 92.7859726,B 4.34323788,C 2.74902105,S 6,T 18,E1 0.0,E2 0.0,E3 0.0,E4 0.0,E5 0.0,E6 0.0}
DECL FDAT FP2={TOOL_NO 5,BASE_NO 9,IPO_FRAME #BASE,POINT2[] " ",TQ_STATE FALSE}
DECL LDAT LCPDAT1={VEL 2.0,ACC 100.0,APO_DIST 100.0,APO_FAC 50.0,AXIS_VEL 100.0,AXIS_ACC 100.0,ORI_TYP #VAR,CIRC_TYP #BASE,JERK_FAC 50.0,GEAR_JERK 50.0,EXAX_IGN 0}
DECL E6POS XP4={X 193.489243,Y 281.196289,Z 197.739868,A 92.7863464,B 4.34535694,C 2.74913096}
DECL FDAT FP4={TOOL_NO 5,BASE_NO 9,IPO_FRAME #BASE,POINT2[] " ",TQ_STATE FALSE}
DECL LDAT LCPDAT3={VEL 1.0,ACC 100.0,APO_DIST 100.0,APO_FAC 50.0,AXIS_VEL 100.0,AXIS_ACC 100.0,ORI_TYP #VAR,CIRC_TYP #BASE,JERK_FAC 50.0,GEAR_JERK 50.0,EXAX_IGN 0}
DECL E6POS XP5={X 342.671112,Y 72.4182281,Z -139.308807,A -50.8470612,B -89.0542603,C -36.8499908,S 6,T 18,E1 0.0,E2 0.0,E3 0.0,E4 0.0,E5 0.0,E6 0.0}
DECL FDAT FP5={TOOL_NO 5,BASE_NO 10,IPO_FRAME #BASE,POINT2[] " ",TQ_STATE FALSE}
DECL PDAT PPDAT2={VEL 100.0,ACC 100.0,APO_DIST 100.0,APO_MODE #CDIS,GEAR_JERK 50.0}
DECL E6POS XP6={X 343.593414,Y 71.2833023,Z -50.6105003,A -10.3100405,B -86.5372467,C -77.3689117,S 6,T 18,E1 0.0,E2 0.0,E3 0.0,E4 0.0,E5 0.0,E6 0.0}
DECL FDAT FP6={TOOL_NO 5,BASE_NO 10,IPO_FRAME #BASE,POINT2[] " ",TQ_STATE FALSE}
DECL LDAT LCPDAT6={VEL 1.0,ACC 100.0,APO_DIST 100.0,APO_FAC 50.0,AXIS_VEL 100.0,AXIS_ACC 100.0,ORI_TYP #VAR,CIRC_TYP #BASE,JERK_FAC 50.0,GEAR_JERK 50.0,EXAX_IGN 0}
DECL E6POS XP7={X 347.644989,Y 161.104599,Z -44.6483192,A -19.0984497,B -87.3924408,C -68.7215729,S 6,T 18,E1 0.0,E2 0.0,E3 0.0,E4 0.0,E5 0.0,E6 0.0}
DECL FDAT FP7={TOOL_NO 5,BASE_NO 10,IPO_FRAME #BASE,POINT2[] " ",TQ_STATE FALSE}
DECL LDAT LCPDAT5={VEL 1.0,ACC 100.0,APO_DIST 100.0,APO_FAC 50.0,AXIS_VEL 100.0,AXIS_ACC 100.0,ORI_TYP #VAR,CIRC_TYP #BASE,JERK_FAC 50.0,GEAR_JERK 50.0,EXAX_IGN 0}
DECL LDAT LCPDAT0={VEL 2.0,ACC 100.0,APO_DIST 100.0,APO_FAC 50.0,AXIS_VEL 100.0,AXIS_ACC 100.0,ORI_TYP #VAR,CIRC_TYP #BASE,JERK_FAC 50.0,GEAR_JERK 50.0,EXAX_IGN 0}
DECL LDAT LCPDAT7={VEL 1.0,ACC 100.0,APO_DIST 100.0,APO_FAC 50.0,AXIS_VEL 100.0,AXIS_ACC 100.0,ORI_TYP #VAR,CIRC_TYP #BASE,JERK_FAC 50.0,GEAR_JERK 50.0,EXAX_IGN 0}
DECL E6POS XP8={X 250.825699,Y 68.5500336,Z -156.140106,A -11.6958599,B -87.5133972,C -76.3972168,S 6,T 18,E1 0.0,E2 0.0,E3 0.0,E4 0.0,E5 0.0,E6 0.0}
DECL FDAT FP8={TOOL_NO 5,BASE_NO 10,IPO_FRAME #BASE,POINT2[] " ",TQ_STATE FALSE}
DECL PDAT PPDAT5={VEL 100.0,ACC 100.0,APO_DIST 100.0,APO_MODE #CDIS,GEAR_JERK 50.0}
DECL E6POS XP9={X 248.171906,Y 68.5325623,Z -57.3552895,A -11.7855797,B -87.5131912,C -76.3081131,S 6,T 18,E1 0.0,E2 0.0,E3 0.0,E4 0.0,E5 0.0,E6 0.0}
DECL FDAT FP9={TOOL_NO 5,BASE_NO 10,IPO_FRAME #BASE,POINT2[] " ",TQ_STATE FALSE}
DECL LDAT LCPDAT8={VEL 1.0,ACC 100.0,APO_DIST 100.0,APO_FAC 50.0,AXIS_VEL 100.0,AXIS_ACC 100.0,ORI_TYP #VAR,CIRC_TYP #BASE,JERK_FAC 50.0,GEAR_JERK 50.0,EXAX_IGN 0}
DECL E6POS XP10={X 248.180099,Y 157.122101,Z -57.3562584,A -11.7488298,B -87.5131836,C -76.344368,S 6,T 18,E1 0.0,E2 0.0,E3 0.0,E4 0.0,E5 0.0,E6 0.0}
DECL FDAT FP10={TOOL_NO 5,BASE_NO 10,IPO_FRAME #BASE,POINT2[] " ",TQ_STATE FALSE}
DECL LDAT LCPDAT9={VEL 2.0,ACC 100.0,APO_DIST 100.0,APO_FAC 50.0,AXIS_VEL 100.0,AXIS_ACC 100.0,ORI_TYP #VAR,CIRC_TYP #BASE,JERK_FAC 50.0,GEAR_JERK 50.0,EXAX_IGN 0}
DECL LDAT LCPDAT10={VEL 2.0,ACC 100.0,APO_DIST 100.0,APO_FAC 50.0,AXIS_VEL 100.0,AXIS_ACC 100.0,ORI_TYP #VAR,CIRC_TYP #BASE,JERK_FAC 50.0,GEAR_JERK 50.0,EXAX_IGN 0}
DECL LDAT LCPDAT11={VEL 2.0,ACC 100.0,APO_DIST 100.0,APO_FAC 50.0,AXIS_VEL 100.0,AXIS_ACC 100.0,ORI_TYP #VAR,CIRC_TYP #BASE,JERK_FAC 50.0,GEAR_JERK 50.0,EXAX_IGN 0}
DECL E6POS XP13={X 151.932297,Y 160.193802,Z -51.2728195,A -34.5059509,B -88.7539063,C -53.1838417,S 6,T 18,E1 0.0,E2 0.0,E3 0.0,E4 0.0,E5 0.0,E6 0.0}
DECL FDAT FP13={TOOL_NO 5,BASE_NO 10,IPO_FRAME #BASE,POINT2[] " ",TQ_STATE FALSE}
DECL LDAT LCPDAT13={VEL 2.0,ACC 100.0,APO_DIST 100.0,APO_FAC 50.0,AXIS_VEL 100.0,AXIS_ACC 100.0,ORI_TYP #VAR,CIRC_TYP #BASE,JERK_FAC 50.0,GEAR_JERK 50.0,EXAX_IGN 0}
DECL LDAT LCPDAT14={VEL 2.0,ACC 100.0,APO_DIST 100.0,APO_FAC 50.0,AXIS_VEL 100.0,AXIS_ACC 100.0,ORI_TYP #VAR,CIRC_TYP #BASE,JERK_FAC 50.0,GEAR_JERK 50.0,EXAX_IGN 0}
DECL PDAT PPDAT0={VEL 100.0,ACC 100.0,APO_DIST 100.0,APO_MODE #CDIS,GEAR_JERK 50.0}
DECL E6POS XP0={X 370.350006,Y -40.2177391,Z 70.7605515,A -140.187607,B -20.9161091,C -85.7391586,S 6,T 27,E1 0.0,E2 0.0,E3 0.0,E4 0.0,E5 0.0,E6 0.0}
DECL FDAT FP0={TOOL_NO 5,BASE_NO 9,IPO_FRAME #BASE,POINT2[] " ",TQ_STATE FALSE}
DECL E6POS XP3={X 193.491898,Y 281.194641,Z 4.73327351,A 92.7861786,B 4.34509897,C 2.74875402}
DECL FDAT FP3={TOOL_NO 5,BASE_NO 9,IPO_FRAME #BASE,POINT2[] " ",TQ_STATE FALSE}
DECL LDAT LCPDAT2={VEL 2.0,ACC 100.0,APO_DIST 100.0,APO_FAC 50.0,AXIS_VEL 100.0,AXIS_ACC 100.0,ORI_TYP #VAR,CIRC_TYP #BASE,JERK_FAC 50.0,GEAR_JERK 50.0,EXAX_IGN 0}
DECL E6POS XP20={X 112.129662,Y 189.295181,Z 18.3459053,A 93.2300034,B 1.39999998,C 1.83000004}
DECL FDAT FP20={TOOL_NO 5,BASE_NO 11,IPO_FRAME #BASE,POINT2[] " ",TQ_STATE FALSE}
DECL E6POS XP14={X 366.011963,Y 291.341156,Z 95.9162903,A 96.3636475,B 4.65242004,C 2.64675307}
DECL FDAT FP14={TOOL_NO 5,BASE_NO 9,IPO_FRAME #BASE,POINT2[] " ",TQ_STATE FALSE}
DECL E6POS XP15={X 362.373596,Y 282.951782,Z -1.78855562,A 96.3680573,B 4.63769197,C 2.64578199}
DECL FDAT FP15={TOOL_NO 5,BASE_NO 9,IPO_FRAME #BASE,POINT2[] " ",TQ_STATE FALSE}
DECL E6POS XP16={X 363.755676,Y 203.040726,Z 8.37380028,A 96.368042,B 4.63726902,C 2.6456461}
DECL FDAT FP16={TOOL_NO 5,BASE_NO 9,IPO_FRAME #BASE,POINT2[] " ",TQ_STATE FALSE}
DECL LDAT LCPDAT4={VEL 1.0,ACC 100.0,APO_DIST 100.0,APO_FAC 50.0,AXIS_VEL 100.0,AXIS_ACC 100.0,ORI_TYP #VAR,CIRC_TYP #BASE,JERK_FAC 50.0,GEAR_JERK 50.0,EXAX_IGN 0}
DECL E6POS XP17={X 367.011322,Y 210.592178,Z 96.5099792,A 96.368721,B 4.63736916,C 2.64742398}
DECL FDAT FP17={TOOL_NO 5,BASE_NO 9,IPO_FRAME #BASE,POINT2[] " ",TQ_STATE FALSE}
DECL E6POS XP18={X 122.127205,Y 114.158562,Z 200.154968,A 93.2300034,B 1.39999998,C 1.83000004}
DECL FDAT FP18={TOOL_NO 5,BASE_NO 11,IPO_FRAME #BASE,POINT2[] " ",TQ_STATE FALSE}
DECL PDAT PPDAT3={VEL 100.0,ACC 100.0,APO_DIST 100.0,APO_MODE #CDIS}
DECL E6POS XP19={X 116.635864,Y 109.446121,Z 20.300478,A 93.2300034,B 1.39999998,C 1.83000004}
DECL FDAT FP19={TOOL_NO 5,BASE_NO 11,IPO_FRAME #BASE,POINT2[] " ",TQ_STATE FALSE}
DECL E6POS XP21={X 118.747551,Y 174.045364,Z 198.689041,A 93.2300034,B 1.39999998,C 1.83000004}
DECL FDAT FP21={TOOL_NO 5,BASE_NO 11,IPO_FRAME #BASE,POINT2[] " ",TQ_STATE FALSE}
DECL E6POS XP22={X 723.833801,Y 64.0526733,Z 177.526505,A 93.2305069,B 1.40343297,C 1.82748401,S 6,T 18,E1 0.0,E2 0.0,E3 0.0,E4 0.0,E5 0.0,E6 0.0}
DECL FDAT FP22={TOOL_NO 5,BASE_NO 11,IPO_FRAME #BASE,POINT2[] " ",TQ_STATE FALSE}
DECL PDAT PPDAT4={VEL 100.0,ACC 100.0,APO_DIST 100.0,APO_MODE #CDIS}
DECL E6POS XG3_HOME={X 593.299988,Y -262.559998,Z 438.690002,A 6.36999989,B 2.11999989,C 1.97000003,S 6,T 18,E1 0.0,E2 0.0,E3 0.0,E4 0.0,E5 0.0,E6 0.0}
DECL FDAT FG3_HOME={TOOL_NO 5,BASE_NO 0,IPO_FRAME #BASE,POINT2[] " ",TQ_STATE FALSE}
DECL PDAT PPDAT7={VEL 100.0,ACC 100.0,APO_DIST 100.0,APO_MODE #CDIS,GEAR_JERK 50.0}
DECL E6POS XG4_HOME={X 593.302673,Y -262.559692,Z 438.690887,A 6.37002182,B 2.11970401,C 1.97006202,S 6,T 18,E1 0.0,E2 0.0,E3 0.0,E4 0.0,E5 0.0,E6 0.0}
DECL FDAT FG4_HOME={TOOL_NO 5,BASE_NO 0,IPO_FRAME #BASE,POINT2[] " ",TQ_STATE FALSE}
DECL PDAT PPDAT8={VEL 100,ACC 100,APO_DIST 100,APO_MODE #CPTP}
DECL E6POS XG3_SISTEMA_VISAO={X 0.0,Y 0.0,Z 283.559998,A 93.2300034,B 1.39999998,C 0.0}
DECL FDAT FG3_sistema_visao={TOOL_NO 5,BASE_NO 11,IPO_FRAME #BASE,POINT2[] " ",TQ_STATE FALSE}
DECL PDAT PPDAT9={VEL 100.0,ACC 100.0,APO_DIST 100.0,APO_MODE #CDIS,GEAR_JERK 50.0}
DECL LDAT LCPDAT16={VEL 2.0,ACC 100.0,APO_DIST 100.0,APO_FAC 50.0,AXIS_VEL 100.0,AXIS_ACC 100.0,ORI_TYP #VAR,CIRC_TYP #BASE,JERK_FAC 50.0,GEAR_JERK 50.0,EXAX_IGN 0}
DECL PDAT PPDAT10={VEL 100.0,ACC 100.0,APO_DIST 100.0,APO_MODE #CDIS,GEAR_JERK 50.0}
DECL E6POS XPVISAO={X 68.3081436,Y 10.0300102,Z 283.573792,A 93.2279434,B 1.39993095,C 0.0838164687,S 6,T 26,E1 0.0,E2 0.0,E3 0.0,E4 0.0,E5 0.0,E6 0.0}
DECL FDAT FPVisao={TOOL_NO 5,BASE_NO 11,IPO_FRAME #BASE,POINT2[] " ",TQ_STATE FALSE}
DECL PDAT PPDAT11={VEL 100.0,ACC 100.0,APO_DIST 100.0,APO_MODE #CDIS,GEAR_JERK 50.0}
DECL LDAT LCPDAT17={VEL 2.0,ACC 100.0,APO_DIST 100.0,APO_FAC 50.0,AXIS_VEL 100.0,AXIS_ACC 100.0,ORI_TYP #VAR,CIRC_TYP #BASE,JERK_FAC 50.0,GEAR_JERK 50.0,EXAX_IGN 0}
DECL PDAT PPDAT12={VEL 100.0,ACC 100.0,APO_DIST 100.0,APO_MODE #CDIS,GEAR_JERK 50.0}
DECL PDAT PPDAT13={VEL 100.0,ACC 100.0,APO_DIST 100.0,APO_MODE #CDIS,GEAR_JERK 50.0}
DECL PDAT PPDAT14={VEL 100.0,ACC 100.0,APO_DIST 100.0,APO_MODE #CDIS,GEAR_JERK 50.0}
DECL PDAT PPDAT15={VEL 100.0,ACC 100.0,APO_DIST 100.0,APO_MODE #CDIS,GEAR_JERK 50.0}
DECL PDAT PPDAT16={VEL 100.0,ACC 100.0,APO_DIST 100.0,APO_MODE #CDIS,GEAR_JERK 50.0}
DECL PDAT PPDAT17={VEL 100.0,ACC 100.0,APO_DIST 100.0,APO_MODE #CDIS,GEAR_JERK 50.0}
DECL PDAT PPDAT18={VEL 100.0,ACC 100.0,APO_DIST 100.0,APO_MODE #CDIS,GEAR_JERK 50.0}
DECL PDAT PPDAT19={VEL 100.0,ACC 100.0,APO_DIST 100.0,APO_MODE #CDIS,GEAR_JERK 50.0}
DECL PDAT PPDAT20={VEL 100.0,ACC 100.0,APO_DIST 100.0,APO_MODE #CDIS,GEAR_JERK 50.0}
DECL PDAT PPDAT21={VEL 100.0,ACC 100.0,APO_DIST 100.0,APO_MODE #CDIS,GEAR_JERK 50.0}
DECL PDAT PPDAT22={VEL 100.0,ACC 100.0,APO_DIST 100.0,APO_MODE #CDIS,GEAR_JERK 50.0}
ENDDAT
